TYPE EC001 :
    STRUCT
    {attribute addProperty Name "A1"}
    A1 : EL1008;
    {attribute addProperty Name "A10"}
    A10 : EL2008;
END_STRUCT
END_TYPE

(* stored: Version 1.1.0.1, ProductVersion 3.1.4024.9
   DUT EC001: Id {88b7d664-8900-036e-3874-96016a870d5c} *)
